// TIA Portal V20 export
DATA_BLOCK "dStruct_Pos16"   // DB30141
{ S7_Optimized_Access := 'TRUE' }
// stored: AutoNumber false, MemoryReserve 100
   VAR
      Axis_Control_Data : Array[0..10] of Struct
         I_SS_bHome : Bool;   // 原点传感器
         I_SS_bFW : Bool;   // 前限位
         I_SS_bBW : Bool;   // 后限位
         I_CMD_bEnableAxis : Bool;   // 使能
         I_CMD_bResetAxis : Bool;   // 复位
         I_CMD_bjogForward : Bool;   // Taster Aufwärts / 正点
         I_CMD_bjogBackward : Bool;   // Taster Abwärts / 反点
         I_CMD_bmoveVelocity : Bool;   // 速度运行
         I_CMD_bstop : Bool;   // 停止
         I_CMD_bfastStop : Bool;   // 急停
         I_CMD_bHoming : Bool;   // 回零
         I_CMD_bGoToPos : Array[0..15] of Bool;   // Start Aufwärts in Automatik / 16个定位
         I_CMD_iGoToPos : Word;   // 16个定位 Word
         I_CMD_bCallAbsPos : Bool;   // 定位位置切换时，单独的定位按钮
         I_CMD_bRelPos : Bool;   // 相对定位
         I_CMD_MyBool : Array[0..5] of Bool;   // 临时变量
         I_Para_rJog_Speed : Array[0..2] of LReal;   // 点动速度/ACC/DEC/JERK
         I_Para_rMV_Speed : Array[0..2] of LReal;   // 速度运行速度/ACC/DEC/JERK
         I_Para_rStop_Dec : Array[0..1] of LReal;   // 速度运行速度/ACC/DEC/JERK
         I_Para_rEStop_Dec : Array[0..1] of LReal;   // 速度运行速度/ACC/DEC/JERK
         I_Para_iNum_Abspos : Int;
         I_Para_rPos_Abs : Array[0..16] of LReal;   // 绝对定位目标位置
         I_Para_rSpeed_Abs : Array[0..16] of LReal;   // Endlage Unten / 绝对定位速度
         I_Para_rAcc_Set : Array[0..16] of LReal;   // 绝对定位加速度
         I_Para_rDec_Set : Array[0..16] of LReal;   // 绝对定位减速度
         I_Para_rJerk_Set : Array[0..16] of LReal;   // 绝对定位加加速度
         I_Para_rSpeedPercent : LReal;   // Endlage Unten / 速度设定百分比
         I_Para_iHomeMode : Int;   // 回零方式
         I_Para_rHomePos : LReal;   // 回零位置
         O_Status_bAxisReady : Bool;   // 轴通讯正常
         O_Status_bAxisEnabled : Bool;   // 轴使能
         O_Status_bjogForward : Bool;   // 轴正点中
         O_Status_bjogBackward : Bool;   // 轴反点中
         O_Status_bHomed : Bool;   // 轴归零完成
         O_Status_bAtHome : Bool;   // 轴在零位
         O_Status_bSstill : Bool;   // 轴静止
         O_Status_bAxisBusy : Bool;   // 轴运行中
         O_Status_bAxisSyned : Bool;   // 同步上
         O_Status_bAxisError : Bool;   // 轴报警
         O_Status_bAtPos : Array[0..15] of Bool;   // Ausgang Aufwärts / 在目标位置上
         O_Status_bPosDone : Array[0..15] of Bool;   // 定位完成
         O_Status_bPosing : Array[0..15] of Bool;   // Ausgang Aufwärts / 定位中
         O_Status_bRelPosDone : Bool;   // 相对定位完成
         O_Status_rActPos : LReal;   // 实际位置
         O_Status_rActSpeed : LReal;   // 实际速度
         O_Status_iAxisFaultNum : UDInt;   // 轴报警代码
         O_Status_iDriveFaultNum : UDInt;   // 驱动报警代码
         O_Status_iFBStatus : Word;   // 运动功能块状态
         O_Status_iMCStatus : Word;   // 运动指令状态
         O_Status_rDriveTorque : LReal;   // 驱动扭矩
         O_Status_rDriveTemp : LReal;   // 驱动温度
         O_Status_rDriveRpm : LReal;   // 驱动转速
         O_Status_AxisName : WString[24];   // Name of axis
         O_Status_mybool : Array[0..5] of Bool;   // 备用
         O_Status_myLreal : Array[0..5] of LReal;   // 备用
         I_InLock_bEnableAxis : Bool;   // 使能
         I_InLock_bResetAxis : Bool;   // 复位
         I_InLock_bjogForward : Bool;   // Taster Aufwärts / 正点
         I_InLock_bjogBackward : Bool;   // Taster Abwärts / 反点
         I_InLock_bmoveVelocity : Bool;   // 速度运行
         I_InLock_bstop : Bool;   // 停止
         I_InLock_bfastStop : Bool;   // 急停
         I_InLock_bHoming : Bool;   // 回零
         I_InLock_bGoToPos : Array[0..16] of Bool;   // Start Aufwärts in Automatik / 16个定位
         I_InLock_iGoToPos : Word;   // 16个定位 Word
         I_InLock_bCallAbsPos : Bool;   // 定位位置切换时，单独的定位按钮
         I_InLock_bRelPos : Bool;   // 相对定位
         I_InLock_MyBool : Array[0..5] of Bool;   // 临时变量
         I_HMI_bEnableAxis : Bool;   // 使能
         I_HMI_bResetAxis : Bool;   // 复位
         I_HMI_bjogForward : Bool;   // Taster Aufwärts / 正点
         I_HMI_bjogBackward : Bool;   // Taster Abwärts / 反点
         I_HMI_bmoveVelocity : Bool;   // 速度运行
         I_HMI_bstop : Bool;   // 停止
         I_HMI_bfastStop : Bool;   // 急停
         I_HMI_bHoming : Bool;   // 回零
         I_HMI_bGoToPos : Array[0..16] of Bool;   // Start Aufwärts in Automatik / 16个定位
         I_HMI_iGoToPos : Word;   // 16个定位 Word
         I_HMI_bCallAbsPos : Bool;   // 定位位置切换时，单独的定位按钮
         I_HMI_bRelPos : Bool;   // 相对定位
         I_HMI_MyBool : Array[0..5] of Bool;   // 临时变量
         I_CDM_bGoToPos_0 : Bool;   // Start Aufwärts in Automatik / 16个定位自动
         I_InLock_bGoToPos_0 : Bool;   // Start Aufwärts in Automatik / 16个定位条件
         I_HMI_bGoToPos_0 : Bool;   // Start Aufwärts in Automatik / 16个定位HMI
         I_CDM_bGoToPos_1 : Bool;   // Start Aufwärts in Automatik / 16个定位自动
         I_InLock_bGoToPos_1 : Bool;   // Start Aufwärts in Automatik / 16个定位条件
         I_HMI_bGoToPos_1 : Bool;   // Start Aufwärts in Automatik / 16个定位HMI
         I_CDM_bGoToPos_2 : Bool;   // Start Aufwärts in Automatik / 16个定位自动
         I_InLock_bGoToPos_2 : Bool;   // Start Aufwärts in Automatik / 16个定位条件
         I_HMI_bGoToPos_2 : Bool;   // Start Aufwärts in Automatik / 16个定位HMI
         I_CDM_bGoToPos_3 : Bool;   // Start Aufwärts in Automatik / 16个定位自动
         I_InLock_bGoToPos_3 : Bool;   // Start Aufwärts in Automatik / 16个定位条件
         I_HMI_bGoToPos_3 : Bool;   // Start Aufwärts in Automatik / 16个定位HMI
         I_CDM_bGoToPos_4 : Bool;   // Start Aufwärts in Automatik / 16个定位自动
         I_InLock_bGoToPos_4 : Bool;   // Start Aufwärts in Automatik / 16个定位条件
         I_HMI_bGoToPos_4 : Bool;   // Start Aufwärts in Automatik / 16个定位HMI
         I_CDM_bGoToPos_5 : Bool;   // Start Aufwärts in Automatik / 16个定位自动
         I_InLock_bGoToPos_5 : Bool;   // Start Aufwärts in Automatik / 16个定位条件
         I_HMI_bGoToPos_5 : Bool;   // Start Aufwärts in Automatik / 16个定位HMI
         I_CDM_bGoToPos_6 : Bool;   // Start Aufwärts in Automatik / 16个定位自动
         I_InLock_bGoToPos_6 : Bool;   // Start Aufwärts in Automatik / 16个定位条件
         I_HMI_bGoToPos_6 : Bool;   // Start Aufwärts in Automatik / 16个定位HMI
         I_CDM_bGoToPos_7 : Bool;   // Start Aufwärts in Automatik / 16个定位自动
         I_InLock_bGoToPos_7 : Bool;   // Start Aufwärts in Automatik / 16个定位条件
         I_HMI_bGoToPos_7 : Bool;   // Start Aufwärts in Automatik / 16个定位HMI
         I_CDM_bGoToPos_8 : Bool;   // Start Aufwärts in Automatik / 16个定位自动
         I_InLock_bGoToPos_8 : Bool;   // Start Aufwärts in Automatik / 16个定位条件
         I_HMI_bGoToPos_8 : Bool;   // Start Aufwärts in Automatik / 16个定位HMI
      END_STRUCT;
      gs_AxisPos16 { S7_SetPoint := 'True'} : Array[0..9] of "sPos16";
   END_VAR
BEGIN
   Axis_Control_Data[0].I_SS_bFW := TRUE;
   Axis_Control_Data[0].I_SS_bBW := TRUE;
   Axis_Control_Data[0].I_Para_rJog_Speed[0] := 10.0;
   Axis_Control_Data[0].I_Para_rJog_Speed[1..2] := 30.0;
   Axis_Control_Data[0].I_Para_rMV_Speed[0] := 20.0;
   Axis_Control_Data[0].I_Para_rMV_Speed[1..2] := 30.0;
   Axis_Control_Data[0].I_Para_rStop_Dec[0] := 30.0;
   Axis_Control_Data[0].I_Para_rStop_Dec[1] := 50.0;
   Axis_Control_Data[0].I_Para_rEStop_Dec[0..1] := 50.0;
   Axis_Control_Data[0].I_Para_iNum_Abspos := 4;
   Axis_Control_Data[0].I_Para_rPos_Abs[1] := 10.0;
   Axis_Control_Data[0].I_Para_rPos_Abs[2] := 20.0;
   Axis_Control_Data[0].I_Para_rPos_Abs[3] := 30.0;
   Axis_Control_Data[0].I_Para_rPos_Abs[4] := 40.0;
   Axis_Control_Data[0].I_Para_rPos_Abs[5] := 50.0;
   Axis_Control_Data[0].I_Para_rPos_Abs[6] := 60.0;
   Axis_Control_Data[0].I_Para_rPos_Abs[7] := 70.0;
   Axis_Control_Data[0].I_Para_rPos_Abs[8] := 80.0;
   Axis_Control_Data[0].I_Para_rPos_Abs[9] := 90.0;
   Axis_Control_Data[0].I_Para_rPos_Abs[10] := 100.0;
   Axis_Control_Data[0].I_Para_rPos_Abs[11] := 110.0;
   Axis_Control_Data[0].I_Para_rPos_Abs[12] := 120.0;
   Axis_Control_Data[0].I_Para_rPos_Abs[13] := 130.0;
   Axis_Control_Data[0].I_Para_rPos_Abs[14] := 140.0;
   Axis_Control_Data[0].I_Para_rPos_Abs[15] := 150.0;
   Axis_Control_Data[0].I_Para_rPos_Abs[16] := 160.0;
   Axis_Control_Data[0].I_Para_rSpeed_Abs[0..16] := 20.0;
   Axis_Control_Data[0].I_Para_rAcc_Set[0..16] := 50.0;
   Axis_Control_Data[0].I_Para_rDec_Set[0..16] := 50.0;
   Axis_Control_Data[0].I_Para_rJerk_Set[0..16] := 50.0;
   Axis_Control_Data[0].I_Para_rSpeedPercent := 20.0;
   Axis_Control_Data[0].O_Status_AxisName := WSTRING#'No axis';
END_DATA_BLOCK
